FUNCTION_BLOCK ACMethodBase EXTENDS ACObject IMPLEMENTS IACMethod
VAR_INPUT
END_VAR
VAR_OUTPUT
END_VAR
VAR
END_VAR

PROPERTY ACInitState : ACInitStateEnum
GET
ACInitState := ACInitStateEnum.Unchanged;
END_GET
END_PROPERTY

METHOD FB_postinit
VAR_INPUT
		root : IACVariobatch;
END_VAR
END_METHOD

PROPERTY InstanceID : UDINT
GET
InstanceID := 0;
END_GET
END_PROPERTY

PROPERTY IsValid : BOOL
GET
IsValid := FALSE;
END_GET
END_PROPERTY

END_FUNCTION_BLOCK

(* stored: Version 1.1.0.1, ProductVersion 3.1.4022.7
   POU ACMethodBase: Id {85ac7060-1ece-469d-b6ba-dc9801c7486e}, SpecialFunc None
   Property ACInitState: Id {831582d6-9136-439e-b3b4-31d1f062cafe}
   Get Get: Id {52430745-f6a2-44e9-aa0a-f1348c9885fc}
   Method FB_postinit: Id {a6291b5b-7e6c-4b6d-b5bc-ca6f6de59193}
   Property InstanceID: Id {34b6e2a7-7077-4c28-b952-7041328962bf}
   Get Get: Id {f5da2b1b-1bab-492c-bd5c-71c80fd1af72}
   Property IsValid: Id {133a1595-5623-473e-a7a3-f231599d7111}
   Get Get: Id {89af1a6d-df99-403a-afae-4454632f547c} *)
